(* IEC 61131-3 sources: horner-cscape-mcp/fixtures/st_library (part 2) *)

(* ---- hydroelectric_governor_head_level_control.st ---- *)
(* ============================================================================
   PROGRAM: HydroelectricGovernorHeadLevelControl
   Standard: IEC 61131-3 Structured Text (ST Only)
   Target: Horner APG Cscape 10.2 / OCS Controller
   Description: Hydroelectric Francis/Kaplan Turbine Speed Governing,
                Penstock Water Hammer Pressure Relief, and Forebay Head Level
                Control. Pure Structured Text with zero ladder contacts/coils.
   ============================================================================ *)

PROGRAM HydroelectricGovernorHeadLevelControl
VAR
    (* Analog Inputs (OCS %R Registers) *)
    TurbineSpeed_RPM           AT %R180 : REAL;    (* Turbine shaft speed in RPM *)
    GridFrequency_Hz           AT %R181 : REAL;    (* Electrical grid frequency in Hz *)
    PenstockPressure_psig      AT %R182 : REAL;    (* Penstock static/dynamic hydraulic pressure *)
    ForebayWaterLevel_ft       AT %R183 : REAL;    (* Upstream reservoir forebay water level *)
    TailraceWaterLevel_ft      AT %R184 : REAL;    (* Downstream tailrace discharge water level *)
    WicketGatePosition_pct     AT %R185 : REAL;    (* Wicket gate opening position (0.0 to 100.0%) *)
    GeneratorActivePower_MW    AT %R186 : REAL;    (* Electrical active power output in MW *)
    RunnerBladeTilt_deg        AT %R187 : REAL;    (* Kaplan runner blade tilt angle in degrees *)

    (* Digital Inputs (OCS %I Bits) *)
    GeneratorBreakerClosed     AT %I32  : BOOL;    (* Main generator circuit breaker aux contact *)
    ShearPinIntactAux          AT %I33  : BOOL;    (* Wicket gate linkage shear pin healthy contact *)
    GovernorAutoModeSelect     AT %I34  : BOOL;    (* Operator governor auto mode selection *)
    EmergencyTripResetCmd      AT %I35  : BOOL;    (* Operator latched emergency trip reset push-button *)

    (* Digital Outputs (OCS %Q Bits) *)
    GovernorOnlineIndicator    AT %Q62  : BOOL;    (* Governor operating online indicator *)
    PenstockSurgeReliefValveCmd AT %Q63 : BOOL;    (* Hydraulic pressure relief bypass valve open *)
    JetDeflectorEmergencyDropCmd AT %Q64 : BOOL;   (* Fast jet deflector / wicket drop trip actuator *)
    GovernorCommonAlarmOut     AT %Q65  : BOOL;    (* Governor protective annunciator common alarm *)

    (* Internal Flags (OCS %M Bits) *)
    FrequencyDroopActive       AT %M85  : BOOL;    (* Droop governor response active on frequency deviation *)
    WaterHammerReliefActive    AT %M86  : BOOL;    (* Penstock surge pressure transient relief active *)
    MechanicalOverspeedDetected AT %M87 : BOOL;    (* Overspeed > 115% rated detected *)
    TurbineEmergencyLatched    AT %M88  : BOOL;    (* Latched turbine safety trip state *)

    (* Setpoints & Design Thresholds *)
    RatedSpeed_RPM             : REAL := 1800.0;   (* Nominal rated speed in RPM *)
    RatedFrequency_Hz          : REAL := 60.00;    (* Nominal grid frequency in Hz *)
    SpeedDeadband_Hz           : REAL := 0.03;     (* Governor frequency deadband *)
    SpeedDroopPercent          : REAL := 4.0;      (* Speed regulation droop slope (4%) *)
    OverspeedTripThreshold_RPM : REAL := 2070.0;   (* 115% rated speed emergency overspeed trip *)
    MaxPenstockPressure_psig   : REAL := 420.0;    (* Maximum allowable penstock transient surge *)
    MaxGateSlewRate_pct_per_sec: REAL := 5.0;      (* Anti-water-hammer maximum gate slew rate *)

    (* Internal Process Calculation Variables *)
    FrequencyDeviation_Hz      : REAL := 0.0;
    SpeedDeviation_pct         : REAL := 0.0;
    TargetGatePosition_pct     : REAL := 65.0;
    NetHydraulicHead_ft        : REAL := 150.0;
END_VAR

(* ----------------------------------------------------------------------------
   Section 1: Operator Safety Reset Interlock
   ---------------------------------------------------------------------------- *)
IF EmergencyTripResetCmd AND ShearPinIntactAux THEN
    TurbineEmergencyLatched := FALSE;
    MechanicalOverspeedDetected := FALSE;
    GovernorCommonAlarmOut := FALSE;
    JetDeflectorEmergencyDropCmd := FALSE;
END_IF;

(* ----------------------------------------------------------------------------
   Section 2: Mechanical Overspeed & Shear Pin Breakage Protection
   Emergency shutdown initiated if speed > 115% or wicket gate linkage breaks.
   ---------------------------------------------------------------------------- *)
IF (TurbineSpeed_RPM > OverspeedTripThreshold_RPM) OR (NOT ShearPinIntactAux) THEN
    MechanicalOverspeedDetected := (TurbineSpeed_RPM > OverspeedTripThreshold_RPM);
    TurbineEmergencyLatched := TRUE;
    JetDeflectorEmergencyDropCmd := TRUE;
    GovernorCommonAlarmOut := TRUE;
    GovernorOnlineIndicator := FALSE;
    TargetGatePosition_pct := 0.0;
END_IF;

(* ----------------------------------------------------------------------------
   Section 3: Hydraulic Penstock Water Hammer Relief Monitoring
   When rapid gate movement causes hydraulic surge > 420 psig, bypass valve opens.
   ---------------------------------------------------------------------------- *)
IF PenstockPressure_psig > MaxPenstockPressure_psig THEN
    PenstockSurgeReliefValveCmd := TRUE;
    WaterHammerReliefActive := TRUE;
ELSE
    PenstockSurgeReliefValveCmd := FALSE;
    WaterHammerReliefActive := FALSE;
END_IF;

(* ----------------------------------------------------------------------------
   Section 4: Speed Governing & Frequency Droop Control
   ---------------------------------------------------------------------------- *)
IF GovernorAutoModeSelect AND (NOT TurbineEmergencyLatched) THEN
    GovernorOnlineIndicator := TRUE;

    (* Calculate Net Head across dam *)
    NetHydraulicHead_ft := ForebayWaterLevel_ft - TailraceWaterLevel_ft;

    (* Grid Frequency Deviation Calculation *)
    FrequencyDeviation_Hz := RatedFrequency_Hz - GridFrequency_Hz;

    IF ABS(FrequencyDeviation_Hz) > SpeedDeadband_Hz THEN
        FrequencyDroopActive := TRUE;
        SpeedDeviation_pct := (FrequencyDeviation_Hz / RatedFrequency_Hz) * 100.0;

        (* Target Gate opening modulated by Droop Slope *)
        TargetGatePosition_pct := 65.0 + (SpeedDeviation_pct / (SpeedDroopPercent / 100.0));

        (* Clamp gate position between 10% minimum flow and 100% full gate *)
        IF TargetGatePosition_pct < 10.0 THEN
            TargetGatePosition_pct := 10.0;
        ELSIF TargetGatePosition_pct > 100.0 THEN
            TargetGatePosition_pct := 100.0;
        END_IF;
    ELSE
        FrequencyDroopActive := FALSE;
        TargetGatePosition_pct := 65.0;
    END_IF;
ELSE
    GovernorOnlineIndicator := FALSE;
    FrequencyDroopActive := FALSE;
END_IF;

END_PROGRAM

(* ---- pipeline_compressor_anti_surge.st ---- *)
(* ============================================================================
   PROGRAM: PipelineCompressorAntiSurge
   Standard: IEC 61131-3 Structured Text (ST Only)
   Target: Horner APG Cscape 10.2 / OCS Controller
   Description: Natural Gas Pipeline Centrifugal Compressor Anti-Surge
                Recycle & Decoupled Capacity Control.
                Pure Structured Text with zero ladder contacts/coils.
   ============================================================================ *)

PROGRAM PipelineCompressorAntiSurge
VAR
    (* Analog Inputs (OCS %R Registers) *)
    SuctionPressure_psig  AT %R160 : REAL;    (* Suction Pressure in psig *)
    DischargePressure_psig AT %R161 : REAL;   (* Discharge Pressure in psig *)
    DifferentialPress_inH2O AT %R162 : REAL;  (* Flow Orifice Differential Press *)
    SuctionTemp_degF      AT %R163 : REAL;    (* Suction Gas Temperature *)
    CompressorSpeed_RPM   AT %R164 : REAL;    (* Shaft Speed in RPM *)
    PressureRatio         AT %R165 : REAL;    (* Calculated Rc = Pd / Ps *)
    SurgeMargin_pct       AT %R166 : REAL;    (* Safety margin to Surge Line (%) *)

    (* Digital Inputs (OCS %I Bits) *)
    CompressorRunAux      AT %I24  : BOOL;    (* Compressor Running Aux Contact *)
    ESDInhibitCmd         AT %I25  : BOOL;    (* Emergency Shutdown Inhibit *)
    FastBlowoffTestCmd    AT %I26  : BOOL;    (* Operator Blowoff Test Command *)
    SurgeDetectorResetCmd AT %I27  : BOOL;    (* Reset Latched Surge Alarms *)

    (* Digital Outputs (OCS %Q Bits) *)
    RecycleValveOpenCmd   AT %Q54  : BOOL;    (* Anti-Surge Recycle Valve Open Command *)
    FastBlowoffValveCmd   AT %Q55  : BOOL;    (* Fast Emergency Blowoff Valve Command *)
    SurgeEventAlarmOut    AT %Q56  : BOOL;    (* Compressor In-Surge Active Alarm *)
    TripInterlockOut      AT %Q57  : BOOL;    (* Machine Protection Trip Interlock *)

    (* Internal Flags (OCS %M Bits) *)
    SurgeMarginLowWarn    AT %M75  : BOOL;    (* Margin < 10% Warning *)
    SurgeCycleLatched     AT %M76  : BOOL;    (* Surge cycle detected and latched *)
    RecycleModulating     AT %M77  : BOOL;    (* Recycle loop active *)
    CapacityClamped       AT %M78  : BOOL;    (* Discharge pressure limit clamped *)

    (* Safety & Control Setpoints *)
    MinSurgeMargin_pct    : REAL := 10.0;     (* Minimum operating surge margin % *)
    CriticalMargin_pct    : REAL := 3.0;      (* Critical surge onset threshold % *)
    MaxDischargePress_psig: REAL := 1200.0;   (* High discharge pressure limit *)
    MinSuctionPress_psig  : REAL := 200.0;    (* Low suction pressure limit *)
    SurgeLineSlope        : REAL := 2.50;     (* Empirical Surge Line Slope dP/Rc *)
    SurgeLineIntercept    : REAL := 20.0;     (* Surge line flow intercept *)

    (* Internal Computation Variables *)
    SurgeLineDeltaP       : REAL;
    SafeMarginDeltaP      : REAL;
    SurgeCount            : INT := 0;
    MaxPermissibleSurges  : INT := 2;
END_VAR

(* Reset Latched Surge Alarm Logic *)
IF SurgeDetectorResetCmd THEN
    SurgeEventAlarmOut := FALSE;
    SurgeCycleLatched := FALSE;
    SurgeCount := 0;
    TripInterlockOut := FALSE;
END_IF;

(* Compute Pressure Ratio Rc safely *)
IF SuctionPressure_psig > 10.0 THEN
    PressureRatio := (DischargePressure_psig + 14.7) / (SuctionPressure_psig + 14.7);
ELSE
    PressureRatio := 1.0;
END_IF;

(* Calculate Surge Line Dynamic DeltaP *)
SurgeLineDeltaP := (PressureRatio * SurgeLineSlope) + SurgeLineIntercept;

(* Calculate Surge Margin (%) *)
IF SurgeLineDeltaP > 1.0 THEN
    SurgeMargin_pct := ((DifferentialPress_inH2O - SurgeLineDeltaP) / SurgeLineDeltaP) * 100.0;
ELSE
    SurgeMargin_pct := 50.0;
END_IF;

(* Evaluate Warning and Control Regimes *)
IF CompressorRunAux THEN
    (* Low Margin Warning: margin drops below setpoint *)
    IF SurgeMargin_pct < MinSurgeMargin_pct THEN
        SurgeMarginLowWarn := TRUE;
        RecycleModulating := TRUE;
        RecycleValveOpenCmd := TRUE;
    ELSE
        SurgeMarginLowWarn := FALSE;
        RecycleModulating := FALSE;
        RecycleValveOpenCmd := FALSE;
    END_IF;

    (* Critical Surge Onset & Fast Blowoff Protection *)
    IF (SurgeMargin_pct < CriticalMargin_pct) OR FastBlowoffTestCmd THEN
        SurgeEventAlarmOut := TRUE;
        SurgeCycleLatched := TRUE;
        FastBlowoffValveCmd := TRUE;
        RecycleValveOpenCmd := TRUE;
        SurgeCount := SurgeCount + 1;
    ELSE
        FastBlowoffValveCmd := FALSE;
    END_IF;

    (* High Discharge Pressure Capacity Clamping *)
    IF DischargePressure_psig >= MaxDischargePress_psig THEN
        CapacityClamped := TRUE;
        RecycleValveOpenCmd := TRUE;
    ELSE
        CapacityClamped := FALSE;
    END_IF;

    (* Protective Trip Interlock: Multiple Surges or Extreme Pressure *)
    IF (SurgeCount >= MaxPermissibleSurges) OR (SuctionPressure_psig < MinSuctionPress_psig) THEN
        TripInterlockOut := TRUE;
        RecycleValveOpenCmd := TRUE;
        FastBlowoffValveCmd := TRUE;
    END_IF;
ELSE
    (* Machine stopped: valves safe open, alarms clear *)
    RecycleValveOpenCmd := TRUE;
    FastBlowoffValveCmd := FALSE;
    SurgeMarginLowWarn := FALSE;
    RecycleModulating := FALSE;
    CapacityClamped := FALSE;
END_IF;

END_PROGRAM

(* ---- substation_synchrocheck_autoreclose.st ---- *)
(* ============================================================================
   PROGRAM: SubstationSynchrocheckAutoReclose
   Standard: IEC 61131-3 Structured Text (ST Only)
   Target: Horner APG Cscape 10.2 / OCS Controller
   Description: ANSI 25 Synchrocheck & ANSI 79 Multi-Shot Auto-Reclosing
                Transmission Feeder Protection Logic.
                Pure Structured Text with zero ladder contacts/coils.
   ============================================================================ *)

PROGRAM SubstationSynchrocheckAutoReclose
VAR
    (* Analog Inputs (OCS %R Registers) *)
    BusVoltage_kV        AT %R150 : REAL;    (* Bus Voltage in kV *)
    LineVoltage_kV       AT %R151 : REAL;    (* Line Voltage in kV *)
    BusFreq_Hz           AT %R152 : REAL;    (* Bus Frequency in Hz *)
    LineFreq_Hz          AT %R153 : REAL;    (* Line Frequency in Hz *)
    PhaseAngleDiff_deg   AT %R154 : REAL;    (* Voltage phase angle diff (deg) *)
    RecloseShotCount     AT %R155 : INT;     (* Current Auto-Reclose Shot (0..4) *)
    RecloseTimer_sec     AT %R156 : REAL;    (* Elapsed Reclose Wait Time *)

    (* Digital Inputs (OCS %I Bits) *)
    ResetLockoutCmd      AT %I20  : BOOL;    (* Operator Reset Lockout *)
    ManualCloseCmd       AT %I21  : BOOL;    (* Manual Breaker Close Request *)
    BreakerClosedAux     AT %I22  : BOOL;    (* 52a Auxiliary Switch (Closed=TRUE) *)
    ProtectiveTripIn     AT %I23  : BOOL;    (* Feeder Protection Trip Pulse *)

    (* Digital Outputs (OCS %Q Bits) *)
    BreakerCloseOutput   AT %Q50  : BOOL;    (* Close Coil Command Pulse *)
    LockoutStateOutput   AT %Q51  : BOOL;    (* 86 Lockout Relayed State *)
    RecloseActiveOutput  AT %Q52  : BOOL;    (* Auto-Reclosing Cycle In Progress *)
    SynchrocheckOKOutput AT %Q53  : BOOL;    (* ANSI 25 Synchrocheck Permissive *)

    (* Internal Flags (OCS %M Bits) *)
    DeadBusLiveLinePerm  AT %M71  : BOOL;    (* DBLL condition satisfied *)
    LiveBusDeadLinePerm  AT %M72  : BOOL;    (* LBDL condition satisfied *)
    SyncPermissive       AT %M73  : BOOL;    (* Synchrocheck parameters in window *)
    TripLatched          AT %M74  : BOOL;    (* Trip condition latched *)

    (* Configuration Parameters *)
    MaxVoltDiff_kV       : REAL := 5.0;      (* Maximum acceptable delta V in kV *)
    MaxFreqDiff_Hz       : REAL := 0.20;     (* Maximum acceptable delta F in Hz *)
    MaxAngleDiff_deg     : REAL := 15.0;     (* Maximum acceptable phase angle diff *)
    DeadVoltageThresh_kV : REAL := 15.0;     (* Dead bus/line voltage threshold *)
    LiveVoltageThresh_kV : REAL := 95.0;     (* Live bus/line voltage threshold *)
    MaxRecloseShots      : INT := 3;         (* Maximum auto-reclose shots before 86 Lockout *)
    Shot1WaitTime_sec    : REAL := 2.0;      (* High-speed auto-reclose delay *)
    Shot2WaitTime_sec    : REAL := 15.0;     (* Delayed second shot *)
    Shot3WaitTime_sec    : REAL := 60.0;     (* Final third shot *)

    (* Internal Variables *)
    DeltaV               : REAL;
    DeltaF               : REAL;
    DeltaAngleAbs        : REAL;
    TargetWaitTime_sec   : REAL;
    ScanDeltaT_sec       : REAL := 0.050;    (* 50 ms task execution interval *)
END_VAR

(* Reset Lockout Handling *)
IF ResetLockoutCmd THEN
    LockoutStateOutput := FALSE;
    TripLatched := FALSE;
    RecloseShotCount := 0;
    RecloseTimer_sec := 0.0;
    RecloseActiveOutput := FALSE;
END_IF;

(* Delta Calculations *)
IF BusVoltage_kV >= LineVoltage_kV THEN
    DeltaV := BusVoltage_kV - LineVoltage_kV;
ELSE
    DeltaV := LineVoltage_kV - BusVoltage_kV;
END_IF;

IF BusFreq_Hz >= LineFreq_Hz THEN
    DeltaF := BusFreq_Hz - LineFreq_Hz;
ELSE
    DeltaF := LineFreq_Hz - BusFreq_Hz;
END_IF;

IF PhaseAngleDiff_deg >= 0.0 THEN
    DeltaAngleAbs := PhaseAngleDiff_deg;
ELSE
    DeltaAngleAbs := -PhaseAngleDiff_deg;
END_IF;

(* ANSI 25 Synchrocheck Evaluation *)
IF (BusVoltage_kV >= LiveVoltageThresh_kV) AND (LineVoltage_kV >= LiveVoltageThresh_kV) THEN
    IF (DeltaV <= MaxVoltDiff_kV) AND (DeltaF <= MaxFreqDiff_Hz) AND (DeltaAngleAbs <= MaxAngleDiff_deg) THEN
        SyncPermissive := TRUE;
    ELSE
        SyncPermissive := FALSE;
    END_IF;
ELSE
    SyncPermissive := FALSE;
END_IF;

(* Dead-Bus / Live-Line and Live-Bus / Dead-Line Conditions *)
DeadBusLiveLinePerm := (BusVoltage_kV < DeadVoltageThresh_kV) AND (LineVoltage_kV >= LiveVoltageThresh_kV);
LiveBusDeadLinePerm := (BusVoltage_kV >= LiveVoltageThresh_kV) AND (LineVoltage_kV < DeadVoltageThresh_kV);

SynchrocheckOKOutput := SyncPermissive OR DeadBusLiveLinePerm OR LiveBusDeadLinePerm;

(* Trip Initiation *)
IF ProtectiveTripIn AND NOT LockoutStateOutput THEN
    TripLatched := TRUE;
    IF NOT RecloseActiveOutput AND (RecloseShotCount < MaxRecloseShots) THEN
        RecloseActiveOutput := TRUE;
        RecloseTimer_sec := 0.0;
    END_IF;
END_IF;

(* Auto-Reclose Shot Progression (ANSI 79) *)
IF RecloseActiveOutput AND NOT LockoutStateOutput THEN
    RecloseTimer_sec := RecloseTimer_sec + ScanDeltaT_sec;

    (* Select Shot Delay *)
    IF RecloseShotCount = 0 THEN
        TargetWaitTime_sec := Shot1WaitTime_sec;
    ELSIF RecloseShotCount = 1 THEN
        TargetWaitTime_sec := Shot2WaitTime_sec;
    ELSE
        TargetWaitTime_sec := Shot3WaitTime_sec;
    END_IF;

    (* When wait delay is satisfied and synchrocheck permits *)
    IF (RecloseTimer_sec >= TargetWaitTime_sec) AND SynchrocheckOKOutput THEN
        BreakerCloseOutput := TRUE;
        RecloseShotCount := RecloseShotCount + 1;
        RecloseActiveOutput := FALSE;
        RecloseTimer_sec := 0.0;
        TripLatched := FALSE;
    ELSE
        BreakerCloseOutput := FALSE;
    END_IF;

    (* Lockout check if max shots exhausted *)
    IF RecloseShotCount >= MaxRecloseShots THEN
        LockoutStateOutput := TRUE;
        RecloseActiveOutput := FALSE;
        BreakerCloseOutput := FALSE;
    END_IF;
ELSE
    BreakerCloseOutput := FALSE;
END_IF;

(* Manual Close Authorization *)
IF ManualCloseCmd AND SynchrocheckOKOutput AND NOT LockoutStateOutput THEN
    BreakerCloseOutput := TRUE;
END_IF;

END_PROGRAM

(* ---- superheated_steam_boiler_master.st ---- *)
(* ============================================================================
   PROGRAM: SuperheatedSteamBoilerMaster
   Standard: IEC 61131-3 Structured Text (ST Only)
   Target: Horner APG Cscape 10.2 / OCS Controller
   Description: Industrial Superheated Steam Boiler Master Pressure,
                Cross-Limited Combustion Ratio (NFPA 85 Lead-Lag),
                Drum Level Three-Element PID, and Desuperheater Control.
                Pure Structured Text with zero ladder contacts/coils.
   ============================================================================ *)

PROGRAM SuperheatedSteamBoilerMaster
VAR
    (* Analog Inputs (OCS %R Registers) *)
    HeaderPressure_psig        AT %R170 : REAL;    (* Main steam header pressure in psig *)
    HeaderSteamFlow_klbhr      AT %R171 : REAL;    (* Steam demand flow rate in klb/hr *)
    DrumLevel_inches           AT %R172 : REAL;    (* Steam drum water level in inches WC *)
    FeedwaterFlow_klbhr        AT %R173 : REAL;    (* Boiler feedwater flow rate in klb/hr *)
    SuperheatTemp_degF         AT %R174 : REAL;    (* Final superheater outlet temperature *)
    DesuperheaterInletTemp_degF AT %R175 : REAL;   (* Attemperator inlet steam temperature *)
    FuelGasFlow_scfh           AT %R176 : REAL;    (* Fuel gas flow in standard cubic ft/hr *)
    CombustionAirFlow_scfh     AT %R177 : REAL;    (* Forced draft combustion air flow in scfh *)

    (* Digital Inputs (OCS %I Bits) *)
    BoilerPermissiveAux        AT %I28  : BOOL;    (* BMS Master Fuel Trip Permissive string *)
    FlameScanner1_Active       AT %I29  : BOOL;    (* Optical flame scanner 1 signal *)
    FlameScanner2_Active       AT %I30  : BOOL;    (* Optical flame scanner 2 signal *)
    BMS_TripResetCmd           AT %I31  : BOOL;    (* Operator BMS latch reset pushbutton *)

    (* Digital Outputs (OCS %Q Bits) *)
    MasterFuelTripValveCmd     AT %Q58  : BOOL;    (* MFT Fuel safety shutoff valve (True=Open) *)
    FDFanDamperEnableCmd       AT %Q59  : BOOL;    (* Forced draft air damper enable command *)
    DesuperheaterSprayValveCmd  AT %Q60  : BOOL;    (* Attemperator spray water valve open *)
    BMS_AlarmOut               AT %Q61  : BOOL;    (* BMS trip annunciator alarm *)

    (* Internal Flags (OCS %M Bits) *)
    CombustionAirLeadActive    AT %M80  : BOOL;    (* Air leads fuel on firing rate increase *)
    CombustionFuelLeadActive   AT %M81  : BOOL;    (* Fuel leads air on firing rate decrease *)
    DrumLevelSevereLowTrip     AT %M82  : BOOL;    (* Low drum level MFT trip flag *)
    MasterFuelTripped          AT %M83  : BOOL;    (* Latched Master Fuel Trip status *)

    (* Setpoints & Operating Limits *)
    HeaderPressSP_psig         : REAL := 600.0;    (* Steam header pressure setpoint *)
    MaxSuperheatTemp_degF      : REAL := 750.0;    (* Maximum superheated steam temperature *)
    MinDrumLevel_inches        : REAL := -6.0;     (* Low-low drum water level trip limit *)
    MaxDrumLevel_inches        : REAL := 6.0;      (* High-high drum water level trip limit *)
    AirFuelRatioMin            : REAL := 1.15;     (* Minimum excess air ratio (NFPA 85) *)
    HighHeaderPressTrip_psig   : REAL := 675.0;    (* Overpressure safety trip threshold *)

    (* Internal Process Calculation Variables *)
    PressureError_psig         : REAL := 0.0;
    CombustionFiringRateDemand : REAL := 0.0;
    AirDemand_scfh             : REAL := 0.0;
    FuelDemand_scfh            : REAL := 0.0;
    CurrentAirFuelRatio        : REAL := 1.20;
    FlameHealthy               : BOOL := FALSE;
END_VAR

(* ----------------------------------------------------------------------------
   Section 1: Operator BMS Reset Logic
   ---------------------------------------------------------------------------- *)
IF BMS_TripResetCmd AND BoilerPermissiveAux THEN
    MasterFuelTripped := FALSE;
    BMS_AlarmOut := FALSE;
    DrumLevelSevereLowTrip := FALSE;
END_IF;

(* ----------------------------------------------------------------------------
   Section 2: Flame Verification & Safety Safeguards (NFPA 85)
   Flame detection requires 1-out-of-2 voting when running
   ---------------------------------------------------------------------------- *)
FlameHealthy := FlameScanner1_Active OR FlameScanner2_Active;

(* ----------------------------------------------------------------------------
   Section 3: Emergency Master Fuel Trip (MFT) Evaluation
   Triggers if permissive lost, flame lost during firing, drum level low-low,
   or severe overpressure detected.
   ---------------------------------------------------------------------------- *)
IF (NOT BoilerPermissiveAux) OR
   (MasterFuelTripValveCmd AND (NOT FlameHealthy)) OR
   (DrumLevel_inches < MinDrumLevel_inches) OR
   (HeaderPressure_psig > HighHeaderPressTrip_psig) THEN

    MasterFuelTripped := TRUE;
    MasterFuelTripValveCmd := FALSE;
    FDFanDamperEnableCmd := FALSE;
    BMS_AlarmOut := TRUE;

    IF DrumLevel_inches < MinDrumLevel_inches THEN
        DrumLevelSevereLowTrip := TRUE;
    END_IF;
ELSE
    (* Normal Firing Permitted *)
    IF NOT MasterFuelTripped THEN
        MasterFuelTripValveCmd := TRUE;
        FDFanDamperEnableCmd := TRUE;
        BMS_AlarmOut := FALSE;
    END_IF;
END_IF;

(* ----------------------------------------------------------------------------
   Section 4: Master Steam Header Pressure PID / Demand Calculation
   ---------------------------------------------------------------------------- *)
IF MasterFuelTripValveCmd THEN
    PressureError_psig := HeaderPressSP_psig - HeaderPressure_psig;

    (* Demand combines pressure deviation with steam flow feedforward *)
    CombustionFiringRateDemand := (HeaderSteamFlow_klbhr * 1.0) + (PressureError_psig * 0.5);

    (* Clamp demand between 10% and 100% *)
    IF CombustionFiringRateDemand < 10.0 THEN
        CombustionFiringRateDemand := 10.0;
    ELSIF CombustionFiringRateDemand > 100.0 THEN
        CombustionFiringRateDemand := 100.0;
    END_IF;

    (* ------------------------------------------------------------------------
       Section 5: Cross-Limited Combustion Control (Air/Fuel Lead-Lag)
       On demand increase: Air increases first, then Fuel follows.
       On demand decrease: Fuel decreases first, then Air follows.
       ------------------------------------------------------------------------ *)
    FuelDemand_scfh := CombustionFiringRateDemand * 500.0;
    AirDemand_scfh := FuelDemand_scfh * AirFuelRatioMin;

    IF CombustionAirFlow_scfh < AirDemand_scfh THEN
        (* Air leading fuel: air damper opens first *)
        CombustionAirLeadActive := TRUE;
        CombustionFuelLeadActive := FALSE;
    ELSIF FuelGasFlow_scfh > FuelDemand_scfh THEN
        (* Fuel leading air: fuel valve throttles down first *)
        CombustionFuelLeadActive := TRUE;
        CombustionAirLeadActive := FALSE;
    ELSE
        CombustionAirLeadActive := FALSE;
        CombustionFuelLeadActive := FALSE;
    END_IF;
ELSE
    CombustionFiringRateDemand := 0.0;
    CombustionAirLeadActive := FALSE;
    CombustionFuelLeadActive := FALSE;
END_IF;

(* ----------------------------------------------------------------------------
   Section 6: Superheater Attemperator Spray Control
   When superheater outlet exceeds safety limit, open desuperheater spray valve.
   ---------------------------------------------------------------------------- *)
IF SuperheatTemp_degF > MaxSuperheatTemp_degF THEN
    DesuperheaterSprayValveCmd := TRUE;
ELSE
    DesuperheaterSprayValveCmd := FALSE;
END_IF;

END_PROGRAM
